PROGRAM TrafficLight
VAR
	fbTraffic : Traffic; //declaring the function block in the program
	
	iRedColor : INT;  //integers connected with the hmi that control how much time we input
	iYellowColor : INT;
	iGreenColor : INT; 
	
	bRedLight : BOOL; //bool variables that turn the lights on/off through the hmi
	bYellowLight : BOOL;
	bGreenLight : BOOL;
	
	bTurnOn : BOOL; //bool variable that turns the traffic light on/off
	
	bTempActive : BOOL;	// bool variable that sets/resets the time inserted by the user through hmi
	bTextError : BOOL; //bool variable that makes the textbox for error visible/invisible
END_VAR

fbTraffic.iRedIn := iRedColor; //inputing the time durations in the function block's inputs
fbTraffic.iYellowIn := iYellowColor;
fbTraffic.iGreenIn := iGreenColor;

fbTraffic.bActivate := bTempActive; //activating the input for the time duration status

fbTraffic.bStart := bTurnOn; //inputing the status of the traffic light (on/off)

bTextError := fbTraffic.bError;

bRedLight := fbTraffic.bRed; //the bool variables take the status for the lights and switch them on/off accordingly
bYellowLight := fbTraffic.bYellow;
bGreenLight := fbTraffic.bGreen;

fbTraffic(); // calling the function block

END_PROGRAM

(* stored: Version 1.1.0.1, ProductVersion 3.1.4024.12
   POU TrafficLight: Id {2d39c46e-01f1-427b-842b-b95cace55462}, SpecialFunc None *)
